FUNCTION_BLOCK FB_Button
VAR_INPUT
	bIsButtonPressed : BOOL;
END_VAR
VAR_OUTPUT
	bActivate : BOOL;
END_VAR
VAR
	fbToggle_RTRIG : R_TRIG;
END_VAR

// This is a toggle button
fbToggle_RTRIG(clk := bIsButtonPressed);
IF fbToggle_RTRIG.Q THEN
	bActivate := NOT bActivate;
END_IF

END_FUNCTION_BLOCK

(* stored: Version 1.1.0.1, ProductVersion 3.1.4024.12
   POU FB_Button: Id {b2f3118b-ec23-4df5-bd97-034de513c742}, SpecialFunc None *)
